FUNCTION_BLOCK RegisterSkill_HMI (* Service Interface Function Block Type *)
  (* Standard: 61499-2 *)
  (* Version 0.0, 2/13/2024, midxav, template *)
  PACKAGE Main;
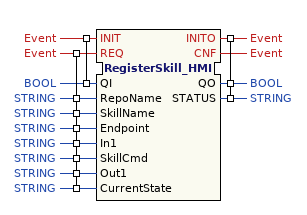
  EVENT_INPUT
    INIT WITH QI;
    REQ WITH RepoName, SkillName, Endpoint, In1, SkillCmd, Out1, CurrentState;
  END_EVENT
  EVENT_OUTPUT
    INITO WITH QO, STATUS;
    CNF;
  END_EVENT
  VAR_INPUT
    QI : BOOL;
    RepoName : STRING;
    SkillName : STRING;
    Endpoint : STRING;
    In1 : STRING;
    SkillCmd : STRING;
    Out1 : STRING;
    CurrentState : STRING;
  END_VAR
  VAR_OUTPUT
    QO : BOOL; (* Event Output Qualifier *)
    STATUS : STRING; (* Service Status *)
  END_VAR
  SERVICE /
    SEQUENCE 
    END_SEQUENCE
  END_SERVICE
END_FUNCTION_BLOCK
